PROGRAM PRG_IsolatedCore
VAR
END_VAR

F_CreateCPULoad();

END_PROGRAM

(* stored: Version 1.1.0.1, ProductVersion 3.1.4026.18
   POU PRG_IsolatedCore: Id {ef03c5c5-9154-4b74-9242-922ea43d0f03}, SpecialFunc None *)
